//{attribute 'qualified_only'}
{attribute 'strict'}
TYPE E_Shapes :
(
	// No shape
	eNoShape := -1,	

	// Triangle
	eTriangle := 0,
	
	// Circle
	eCircle := 1,
	
	// Square
	eSquare := 2
);
END_TYPE

(* stored: Version 1.1.0.1, ProductVersion 3.1.4024.12
   DUT E_Shapes: Id {65947a32-35d0-4dee-882b-85edcf4b5d76} *)
